// TIA Portal V17 export
// export: Created 2023-12-22T15:05:34.4551019Z, ExportSetting WithDefaults, DisplayName Totally Integrated Automation Portal, DisplayVersion V17, DisplayName TIA Portal Openness, DisplayVersion V17, DisplayName TIA Portal Version Control Interface, DisplayVersion V17, DisplayName STEP 7 Professional, DisplayVersion V17, DisplayName STEP 7 Safety, DisplayVersion V17, DisplayName WinCC Advanced, DisplayVersion V17
DATA_BLOCK "Report_Line_2_DB"   // DB52
{ S7_Optimized_Access := 'FALSE' }
VERSION : 0.1
// stored: AutoNumber false, DBAccessibleFromOPCUA true, IsOnlyStoredInLoadMemory false, IsWriteProtectedInAS false
   VAR RETAIN
      Report : Struct
         Last_Day : Int := 3;   // Прошедший день
         Last_Date : Int := 13;   // Прошедшее число (дата)
         Last_Month : Int := 10;   // Прошедший месяц
         RM_1 : Real := 956.8786;   // Расходомер 1
         RM_2 : Real := 0.0;   // Расходомер 2
         D_Mid : Real := 3.0;   // Средняя доза за сутки
         Flow : Real := 17096.32;   // Общая труба (куда происходит дозация)
         Days { S7_SetPoint := 'True'} : Array[1..7] of "Line_Report";   // Дни
         cnt : Int := 7;
         cnt_x : Int := 1;
      END_STRUCT;
      Report_H : "Line_Report";
      Time_DTL : DTL := DTL#2020-10-13-13:05:16.588575848;
   END_VAR
BEGIN
   Report.Days[1].RM_1 := 1936.87;
   Report.Days[2].RM_1 := 2298.9;
   Report.Days[3].RM_1 := 1640.521;
   Report.Days[4].RM_1 := 43.10154;
   Report.Days[5].RM_1 := 5.310862;
   Report.Days[6].RM_1 := 0.0;
   Report.Days[7].RM_1 := 3.251781;
   Report.Days[1..7].RM_2 := 0.0;
   Report.Days[1..7].Res_1 := 0.0;
   Report.Days[1..7].Res_2 := 0.0;
   Report.Days[1].D_Mid := 3.046245;
   Report.Days[2..3].D_Mid := 3.5;
   Report.Days[4].D_Mid := 1.8125;
   Report.Days[5].D_Mid := 4.0;
   Report.Days[6].D_Mid := 0.0;
   Report.Days[7].D_Mid := 3.0;
   Report.Days[1].Flow := 34064.4;
   Report.Days[2].Flow := 35206.3;
   Report.Days[3].Flow := 25124.08;
   Report.Days[4].Flow := 1278.395;
   Report.Days[5].Flow := 77.60835;
   Report.Days[6].Flow := 0.0;
   Report.Days[7].Flow := 58.42366;
   Report.Days[1].WeekDay := 2;
   Report.Days[2].WeekDay := 1;
   Report.Days[3].WeekDay := 7;
   Report.Days[4].WeekDay := 6;
   Report.Days[5].WeekDay := 5;
   Report.Days[6].WeekDay := 4;
   Report.Days[7].WeekDay := 3;
   Report.Days[1].Day := 12;
   Report.Days[2].Day := 11;
   Report.Days[3].Day := 10;
   Report.Days[4].Day := 9;
   Report.Days[5].Day := 8;
   Report.Days[6].Day := 7;
   Report.Days[7].Day := 6;
   Report.Days[1..7].Month := 10;
   Report_H.RM_1 := 0.0;
   Report_H.RM_2 := 0.0;
   Report_H.Res_1 := 15224.0;
   Report_H.Res_2 := 4675.0;
   Report_H.D_Mid := 3.256471;
   Report_H.Flow := 0.0;
   Report_H.WeekDay := 0;
   Report_H.Day := 0;
   Report_H.Month := 0;
END_DATA_BLOCK
